{attribute 'GeneratedUsingTerminal: EL5151-0000-0020'}
{attribute addProperty BoxType "EL5151-0000-0020"}
{attribute addProperty Id "Latch_C_validBOOL1Latch_extern_validBOOL1Set_counter_doneBOOL1Extrapolation_stallBOOL1Status_of_input_ABOOL1Status_of_input_BBOOL1Status_of_input_CBOOL1Status_of_extern_latchBOOL1Sync_errorBOOL1TxPDO_ToggleBOOL1"}
{attribute addProperty CRC "1047478259"}
{attribute addProperty Size "10"}
TYPE Status_3E6F3FF3 :
STRUCT
	{attribute addProperty Name "Latch_C_valid"}
	Latch_C_valid : BOOL;
	{attribute addProperty Name "Latch_extern_valid"}
	Latch_extern_valid : BOOL;
	{attribute addProperty Name "Set_counter_done"}
	Set_counter_done : BOOL;
	{attribute addProperty Name "Extrapolation_stall"}
	Extrapolation_stall : BOOL;
	{attribute addProperty Name "Status_of_input_A"}
	Status_of_input_A : BOOL;
	{attribute addProperty Name "Status_of_input_B"}
	Status_of_input_B : BOOL;
	{attribute addProperty Name "Status_of_input_C"}
	Status_of_input_C : BOOL;
	{attribute addProperty Name "Status_of_extern_latch"}
	Status_of_extern_latch : BOOL;
	{attribute addProperty Name "Sync_error"}
	Sync_error : BOOL;
	{attribute addProperty Name "TxPDO_Toggle"}
	TxPDO_Toggle : BOOL;
END_STRUCT
END_TYPE

(* stored: Version 1.2.0.0, ProductVersion 3.1.4024.9
   DUT Status_3E6F3FF3: Id {05d994fb-049f-4152-98fd-8d4a598992be} *)
